{attribute 'qualified_only'}
{attribute 'strict'}
{attribute 'to_string'}
TYPE E_1026_Set_drive_mode :
(
	Manual_mode := 1,
	Automatic_mode:=2
)UINT;
END_TYPE

(* stored: Version 1.1.0.1, ProductVersion 3.1.4026.17
   DUT E_1026_Set_drive_mode: Id {291b18db-3204-4be2-be6c-995e6bd40fff} *)
